{attribute 'linkalways'} 
{attribute 'no_explicit_call' := 'This FB is a CLASS and must be accessed using methods or properties'}
{attribute 'enable_dynamic_creation'}
FUNCTION_BLOCK FINAL ABS_DINT EXTENDS Node
VAR
	in : _DINT(0);
	out : _DINT(0);
END_VAR

METHOD PUBLIC Clone : I_Node
VAR
	pNode : POINTER TO ABS_DINT;
END_VAR
pNode := __NEW(ABS_DINT);
Clone := pNode^;
END_METHOD

METHOD FB_init : BOOL
VAR_INPUT
	bInitRetains : BOOL; // if TRUE, the retain variables are initialized (warm start / cold start)
	bInCopyCode : BOOL;  // if TRUE, the instance afterwards gets moved into the copy code (online change)
END_VAR
AddInput('in',THIS^.in);
AddOutput('out', THIS^.out);
END_METHOD

METHOD PROTECTED OnExecute
VAR
END_VAR
out.Value := ABS(in.Value);
END_METHOD

END_FUNCTION_BLOCK

(* stored: Version 1.1.0.1, ProductVersion 3.1.4024.15
   POU ABS_DINT: Id {a1a95997-e1e1-4243-ad3b-d862ef43fe70}, SpecialFunc None
   Folder Constructor: Id {1d40ab11-36ab-466f-b346-9eda36fbb358}
   Method Clone: Id {f576971f-ebce-4318-b52b-7c87363a00f0}
   Method FB_init: Id {27348846-4384-4b1d-bc86-28678d510776}
   Method OnExecute: Id {d3532dbf-0194-4e20-b9e6-f54b9a175f77} *)
